FUNCTION_BLOCK SEMAPHORE_BUTTON (* Basic Function Block Type *)
  (* Standard: 61499-2 *)
  (* Version 0.3, 2009-09-15, JHC, Holobloc Inc, Changed transition priorities. *)
  (* Version 0.2, 2003-12-04, JHC, Rockwell Automation, Renamed for better indexing. *)
  (* Version 0.1, 2002-11-05, JHC, Rockwell Automation, Corrected missing ST element in Algorithm REQ. *)
  (* Version 0.0, 2000-05-30, JHC, Rockwell Automation *)
  (* Compiler header: package fb.rt.Assingment; *)
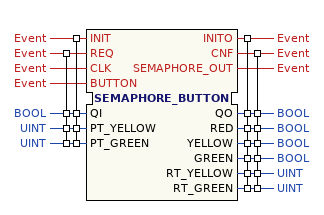
  EVENT_INPUT
    INIT WITH QI, PT_YELLOW, PT_GREEN; (* Initialization Request *)
    REQ WITH QI, PT_YELLOW, PT_GREEN; (* Normal Execution Request *)
    CLK;
    BUTTON;
  END_EVENT
  EVENT_OUTPUT
    INITO WITH QO, RED, YELLOW, GREEN, RT_YELLOW, RT_GREEN; (* Initialization Confirm *)
    CNF WITH YELLOW, RED, QO, GREEN, RT_YELLOW, RT_GREEN; (* Execution Confirmation *)
    SEMAPHORE_OUT;
  END_EVENT
  VAR_INPUT
    QI : BOOL; (* Input event qualifier *)
    PT_YELLOW : UINT;
    PT_GREEN : UINT;
  END_VAR
  VAR_OUTPUT
    QO : BOOL; (* Output event qualifier *)
    RED : BOOL;
    YELLOW : BOOL;
    GREEN : BOOL;
    RT_YELLOW : UINT;
    RT_GREEN : UINT;
  END_VAR
  VAR
    BT_COUNT : UINT;
  END_VAR
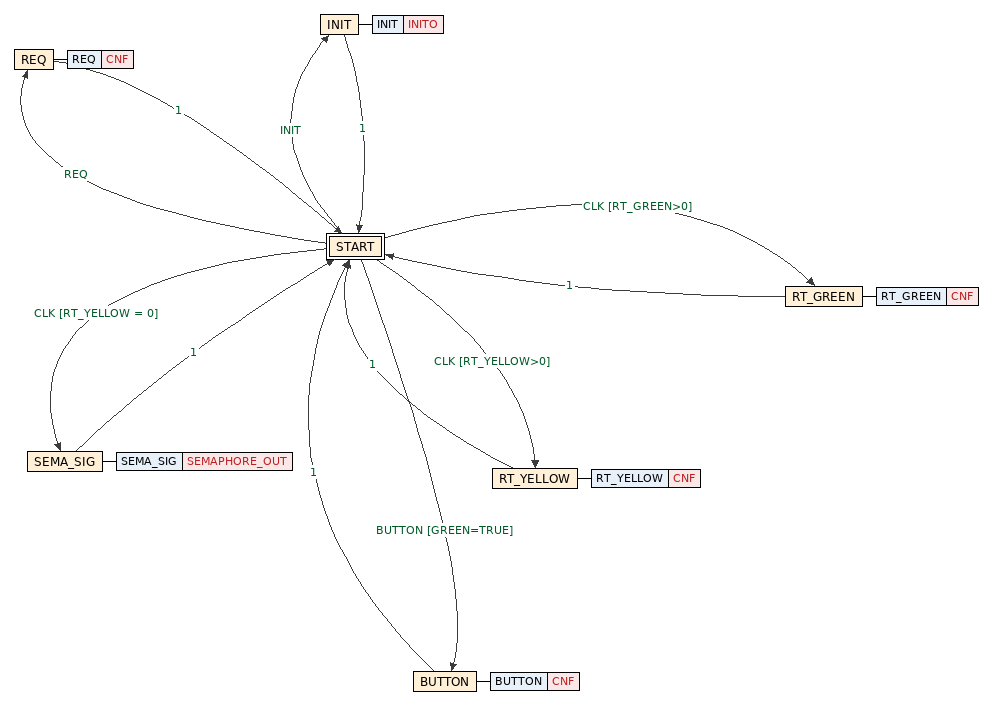
  EC_STATES
    START; (* Initial State *)
    INIT : INIT -> INITO; (* Initialization *)
    REQ : REQ -> CNF; (* Normal execution *)
    RT_GREEN : RT_GREEN -> CNF;
    RT_YELLOW : RT_YELLOW -> CNF;
    SEMA_SIG : SEMA_SIG -> SEMAPHORE_OUT;
    BUTTON : BUTTON -> CNF;
  END_STATES
  EC_TRANSITIONS
    INIT TO START := 1;
    START TO REQ := REQ;
    START TO INIT := INIT;
    REQ TO START := 1;
    START TO RT_GREEN := CLK [RT_GREEN>0];
    RT_GREEN TO START := 1;
    START TO RT_YELLOW := CLK [RT_YELLOW>0];
    RT_YELLOW TO START := 1;
    START TO SEMA_SIG := CLK [RT_YELLOW = 0];
    SEMA_SIG TO START := 1;
    START TO BUTTON := BUTTON [GREEN=TRUE];
    BUTTON TO START := 1;
  END_TRANSITIONS
  ALGORITHM INIT IN ST: (* Initialization algorithm *)

  END_ALGORITHM
  ALGORITHM REQ IN ST: (* Normally executed algorithm *)
RT_GREEN := PT_GREEN;
RT_YELLOW := PT_YELLOW;
BT_COUNT := 4;
RED := FALSE;
YELLOW := FALSE;
GREEN := FALSE;
  END_ALGORITHM
  ALGORITHM RT_GREEN IN ST:
RT_GREEN := RT_GREEN - 1;
GREEN := (RT_GREEN <= PT_GREEN);
GREEN := NOT(RT_GREEN = 0);
  END_ALGORITHM
  ALGORITHM RT_YELLOW IN ST:
RT_YELLOW := RT_YELLOW - 1;
YELLOW := (RT_YELLOW <= PT_YELLOW);
YELLOW := NOT(RT_YELLOW = 0);
RED := (RT_YELLOW = 0);
  END_ALGORITHM
  ALGORITHM SEMA_SIG IN ST:
RED := TRUE;
RT_YELLOW := RT_YELLOW - 1;
  END_ALGORITHM
  ALGORITHM BUTTON IN ST:
IF BT_COUNT > 0  THEN
BT_COUNT := BT_COUNT-1;
END_IF;
IF BT_COUNT = 0  THEN
BT_COUNT := BT_COUNT-1;
RT_GREEN := 4;
RT_YELLOW := PT_YELLOW;
END_IF;
  END_ALGORITHM
END_FUNCTION_BLOCK
